{attribute addProperty BoxType "EL5021-0000-0016"}
{attribute addProperty Id "ControlAT %Q*Control_5DF70A111621Set_counter_valueAT %Q*UDINT32417"}
{attribute addProperty CRC "767388073"}
{attribute addProperty SizeInBites "48"}
{attribute addProperty SizeInBytes "6"}
TYPE ENC_Control_2DBD69A9 :
STRUCT
	{attribute addProperty Name "Control"}
	Control AT %Q* : Control_5DF70A11;
	{attribute addProperty Name "Set_counter_value"}
	Set_counter_value AT %Q* : UDINT;
END_STRUCT
END_TYPE

(* stored: Version 1.2.0.0, ProductVersion 3.1.4024.9
   DUT ENC_Control_2DBD69A9: Id {8ceebd00-8273-4054-8b62-9b0eb9d29f2c} *)
